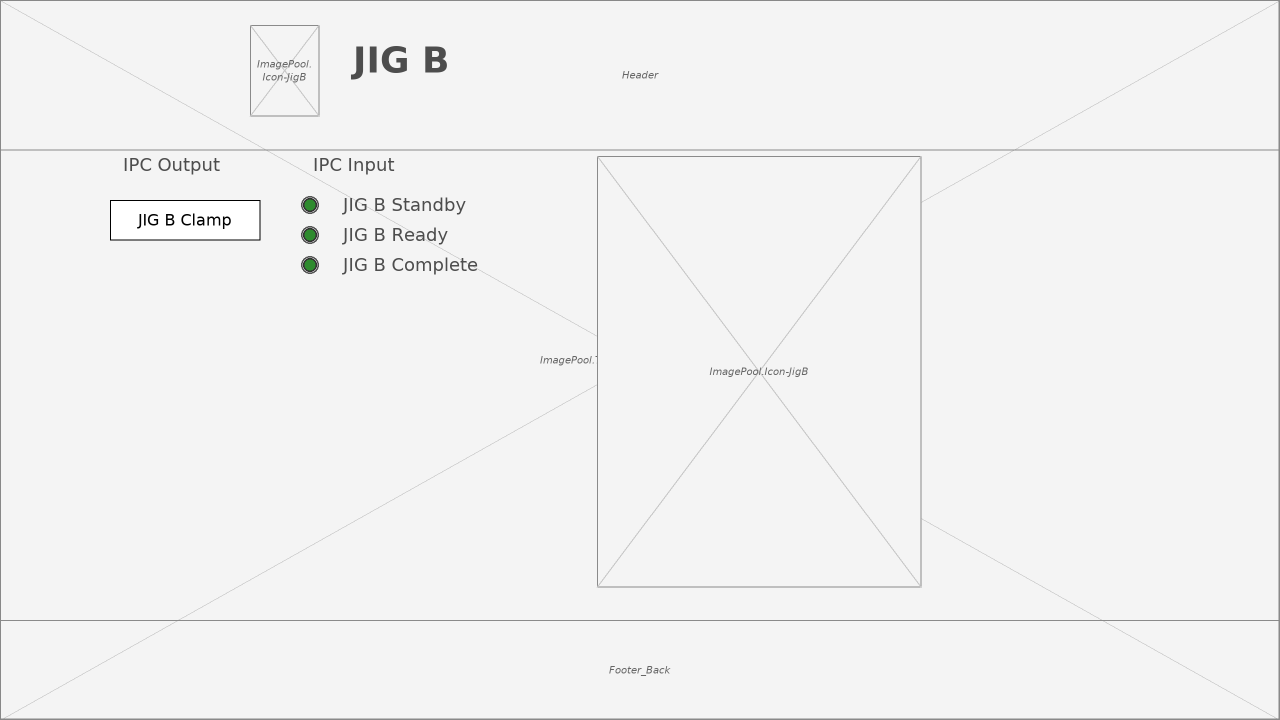
VISUALIZATION PAGE_JIG_B  // 1280x720
    Image (0,0 1280x720), image: ImagePool.The-New-Silver-Backgrounds
    Frame (0,620 1280x100)
        shows Footer_Back()
    Frame (0,0 1280x150)
        shows Header()
    Label (350,40 300x40), "JIG B"
    Label (120,150 150x30), "IPC Output"
    RoundedRectangle (110,200 150x40), "JIG B Clamp"
        toggle GVL.JIGB_Clamp
    Label (310,150 150x30), "IPC Input"
    Label (340,220 170x30), "JIG B Ready"
    Lamp1 (300,225 20x20), variable: GVL.JIGB_Ready, style: Lamp-Lamp1-Green
    Label (340,190 170x30), "JIG B Standby"
    Lamp1 (300,195 20x20), variable: GVL.JIGB_Standby, style: Lamp-Lamp1-Green
    Image (250,25 69x91), image: ImagePool.Icon-JigB
    Image (597,156 324x431), image: ImagePool.Icon-JigB
    Label (340,250 170x30), "JIG B Complete"
    Lamp1 (300,255 20x20), variable: GVL.JIGB_Complete, style: Lamp-Lamp1-Green
END_VISUALIZATION

(* stored: Version 1.1.0.1, ProductVersion 3.1.4024.12
   Visu PAGE_JIG_B: Id {a09d66ac-a526-46b6-84b8-2d614570c632} *)
